(* IEC 61131-3 sources: intralogisticsai/plc_programs, 4 files *)

(* ---- roots_warehouse_simulation.st ---- *)
PROGRAM RootsWarehouseSimulation
  VAR
    (* Physical I/O *)
    emergency_stop AT %IX0.0 : BOOL;
    manual_reset AT %IX0.1 : BOOL;

    (* Process Control Signals - MODBUS 1000-1008 *)
    plc_cycle_stopped AT %QX125.0 : BOOL;
    plc_cycle_running AT %QX125.1 : BOOL;
    pick_error AT %QX125.2 : BOOL;
    pick_to_assembly_in_process AT %QX125.3 : BOOL;
    pick_to_assembly_complete AT %QX125.4 : BOOL;
    pick_to_receiving_in_process AT %QX125.5 : BOOL;
    pick_to_receiving_complete AT %QX125.6 : BOOL;
    pick_to_warehouse_in_process AT %QX125.7 : BOOL;
    pick_to_warehouse_complete AT %QX126.0 : BOOL;

    (* Pick Bin Controls - MODBUS 2000-2011 - ERP Controlled Coils *)
    pick_bin_01 AT %QX250.0 : BOOL;
    pick_bin_02 AT %QX250.1 : BOOL;
    pick_bin_03 AT %QX250.2 : BOOL;
    pick_bin_04 AT %QX250.3 : BOOL;
    pick_bin_05 AT %QX250.4 : BOOL;
    pick_bin_06 AT %QX250.5 : BOOL;
    pick_bin_07 AT %QX250.6 : BOOL;
    pick_bin_08 AT %QX250.7 : BOOL;
    pick_bin_09 AT %QX251.0 : BOOL;
    pick_bin_10 AT %QX251.1 : BOOL;
    pick_bin_11 AT %QX251.2 : BOOL;
    pick_bin_12 AT %QX251.3 : BOOL;

    (* Station Status Controls - MODBUS 2020-2023 - ERP Controlled Coils *)
    to_receiving_sta_1 AT %QX252.4 : BOOL;
    from_receiving_sta_1 AT %QX252.5 : BOOL;
    to_assembly_sta_2 AT %QX252.6 : BOOL;
    from_assembly_sta_2 AT %QX252.7 : BOOL;

    (* Statistics and Monitoring - MODBUS 100-106 *)
    cycle_counter AT %MW100 : INT;
    pick_operations_total AT %MW101 : INT;
    assembly_picks AT %MW102 : INT;
    receiving_picks AT %MW103 : INT;
    warehouse_picks AT %MW104 : INT;
    error_count AT %MW105 : INT;
    uptime_seconds AT %MW106 : INT;
END_VAR

VAR
    (* Internal Variables - No direct addressing *)
    assembly_timer : INT;
    receiving_timer : INT;
    warehouse_timer : INT;
    assembly_complete_timer : INT;
    receiving_complete_timer : INT;
    warehouse_complete_timer : INT;
    any_bin_selected : BOOL;
    assembly_requested : BOOL;
    receiving_requested : BOOL;
    warehouse_requested : BOOL;
    assembly_in_progress : BOOL;
    receiving_in_progress : BOOL;
    warehouse_in_progress : BOOL;
    uptime_timer : INT;
END_VAR

(* Perfect world system - always running, never errors *)
  plc_cycle_running := TRUE;
  plc_cycle_stopped := FALSE;
  pick_error := FALSE;

  (* Increment counters *)
  cycle_counter := cycle_counter + 1;

  (* Uptime calculation - increment every 10 cycles (approximately 1 second at 100ms) *)
  uptime_timer := uptime_timer + 1;
  IF uptime_timer >= 10 THEN
    uptime_timer := 0;
    uptime_seconds := uptime_seconds + 1;
  END_IF;

  (* ERP Command Detection *)
  any_bin_selected := pick_bin_01 OR pick_bin_02 OR pick_bin_03 OR pick_bin_04 OR pick_bin_05 OR pick_bin_06 OR pick_bin_07 OR pick_bin_08 OR pick_bin_09 OR pick_bin_10 OR pick_bin_11 OR pick_bin_12;

  assembly_requested := any_bin_selected AND to_assembly_sta_2;
  receiving_requested := any_bin_selected AND to_receiving_sta_1;
  warehouse_requested := any_bin_selected AND (NOT to_assembly_sta_2) AND (NOT to_receiving_sta_1);

  (* Assembly Operation - 20 Second Robot Simulation *)
  IF assembly_requested AND NOT assembly_in_progress THEN
    (* Start assembly operation *)
    assembly_in_progress := TRUE;
    pick_to_assembly_in_process := TRUE;
    assembly_timer := 0;
  END_IF;

  IF assembly_in_progress THEN
    assembly_timer := assembly_timer + 1;
    IF assembly_timer >= 200 THEN (* 20.0 seconds at 100ms cycles *)
      (* Complete assembly operation *)
      pick_to_assembly_complete := TRUE;
      pick_to_assembly_in_process := FALSE;
      assembly_in_progress := FALSE;
      assembly_timer := 0;
      assembly_picks := assembly_picks + 1;
      pick_operations_total := pick_operations_total + 1;
    END_IF;
  END_IF;

  (* Receiving Operation - 20 Second Robot Simulation *)
  IF receiving_requested AND NOT receiving_in_progress THEN
    (* Start receiving operation *)
    receiving_in_progress := TRUE;
    pick_to_receiving_in_process := TRUE;
    receiving_timer := 0;
  END_IF;

  IF receiving_in_progress THEN
    receiving_timer := receiving_timer + 1;
    IF receiving_timer >= 200 THEN (* 20.0 seconds at 100ms cycles *)
      (* Complete receiving operation *)
      pick_to_receiving_complete := TRUE;
      pick_to_receiving_in_process := FALSE;
      receiving_in_progress := FALSE;
      receiving_timer := 0;
      receiving_picks := receiving_picks + 1;
      pick_operations_total := pick_operations_total + 1;
    END_IF;
  END_IF;

  (* Warehouse Operation - 20 Second Robot Simulation *)
  IF warehouse_requested AND NOT warehouse_in_progress THEN
    (* Start warehouse operation *)
    warehouse_in_progress := TRUE;
    pick_to_warehouse_in_process := TRUE;
    warehouse_timer := 0;
  END_IF;

  IF warehouse_in_progress THEN
    warehouse_timer := warehouse_timer + 1;
    IF warehouse_timer >= 200 THEN (* 20.0 seconds at 100ms cycles *)
      (* Complete warehouse operation *)
      pick_to_warehouse_complete := TRUE;
      pick_to_warehouse_in_process := FALSE;
      warehouse_in_progress := FALSE;
      warehouse_timer := 0;
      warehouse_picks := warehouse_picks + 1;
      pick_operations_total := pick_operations_total + 1;
    END_IF;
  END_IF;

  (* Auto-reset COMPLETE signals after 10 seconds to allow ERP processing time *)
  IF pick_to_assembly_complete THEN
    assembly_complete_timer := assembly_complete_timer + 1;
    IF assembly_complete_timer >= 100 THEN (* 10 seconds *)
      pick_to_assembly_complete := FALSE;
      assembly_complete_timer := 0;
    END_IF;
  ELSE
    assembly_complete_timer := 0;
  END_IF;

  IF pick_to_receiving_complete THEN
    receiving_complete_timer := receiving_complete_timer + 1;
    IF receiving_complete_timer >= 100 THEN (* 10 seconds *)
      pick_to_receiving_complete := FALSE;
      receiving_complete_timer := 0;
    END_IF;
  ELSE
    receiving_complete_timer := 0;
  END_IF;

  IF pick_to_warehouse_complete THEN
    warehouse_complete_timer := warehouse_complete_timer + 1;
    IF warehouse_complete_timer >= 100 THEN (* 10 seconds *)
      pick_to_warehouse_complete := FALSE;
      warehouse_complete_timer := 0;
    END_IF;
  ELSE
    warehouse_complete_timer := 0;
  END_IF;

END_PROGRAM

CONFIGURATION Config0
  RESOURCE Res0 ON PLC
    TASK Main(INTERVAL := T#100ms,PRIORITY := 0);
    PROGRAM Inst0 WITH Main : RootsWarehouseSimulation;
  END_RESOURCE
END_CONFIGURATION

(* ---- simple_modbus_server.st ---- *)
(*
Simple CODESYS Structured Text Program
Intralogistics Learning Lab - Basic MODBUS TCP Server
Provides basic I/O simulation compatible with ERP integration
*)

PROGRAM PLC_PRG
VAR
    (* Conveyor System Variables *)
    Conveyor1_Run: BOOL := FALSE;           (* Address 40001 *)
    Conveyor1_Speed: INT := 0;              (* Address 40002 *)
    Conveyor1_Status: BOOL := FALSE;        (* Address 40003 *)

    Conveyor2_Run: BOOL := FALSE;           (* Address 40004 *)
    Conveyor2_Speed: INT := 0;              (* Address 40005 *)
    Conveyor2_Status: BOOL := FALSE;        (* Address 40006 *)

    (* Storage Robot Variables *)
    Robot_Position_X: INT := 0;             (* Address 40007 *)
    Robot_Position_Y: INT := 0;             (* Address 40008 *)
    Robot_Position_Z: INT := 0;             (* Address 40009 *)
    Robot_Gripper_Open: BOOL := FALSE;      (* Address 40010 *)
    Robot_Busy: BOOL := FALSE;              (* Address 40011 *)

    (* RFID System Variables *)
    RFID_Station1_Active: BOOL := FALSE;    (* Address 40012 *)
    RFID_Station1_TagID: DWORD := 0;        (* Address 40013-40014 *)
    RFID_Station2_Active: BOOL := FALSE;    (* Address 40015 *)
    RFID_Station2_TagID: DWORD := 0;        (* Address 40016-40017 *)

    (* Safety System *)
    Emergency_Stop: BOOL := FALSE;          (* Address 40018 *)
    Safety_OK: BOOL := TRUE;                (* Address 40019 *)
    System_Ready: BOOL := FALSE;            (* Address 40020 *)

    (* Simulation Timers *)
    Cycle_Timer: TIME;
    Robot_Move_Timer: TIME;

    (* Internal simulation variables *)
    Simulation_Active: BOOL := TRUE;
    Cycle_Count: INT := 0;
END_VAR

(* Main Program Logic *)

(* System Ready Logic *)
System_Ready := Safety_OK AND NOT Emergency_Stop;

(* Conveyor Control Logic *)
IF System_Ready THEN
    IF Conveyor1_Run THEN
        Conveyor1_Status := TRUE;
        IF Conveyor1_Speed = 0 THEN
            Conveyor1_Speed := 50;  (* Default speed *)
        END_IF
    ELSE
        Conveyor1_Status := FALSE;
        Conveyor1_Speed := 0;
    END_IF

    IF Conveyor2_Run THEN
        Conveyor2_Status := TRUE;
        IF Conveyor2_Speed = 0 THEN
            Conveyor2_Speed := 50;  (* Default speed *)
        END_IF
    ELSE
        Conveyor2_Status := FALSE;
        Conveyor2_Speed := 0;
    END_IF
ELSE
    (* Emergency stop - halt all conveyors *)
    Conveyor1_Status := FALSE;
    Conveyor1_Speed := 0;
    Conveyor2_Status := FALSE;
    Conveyor2_Speed := 0;
END_IF

(* Robot Simulation Logic *)
IF System_Ready AND NOT Robot_Busy THEN
    (* Simple position simulation *)
    IF Cycle_Count MOD 100 = 0 THEN
        Robot_Position_X := Robot_Position_X + 10;
        IF Robot_Position_X > 1000 THEN
            Robot_Position_X := 0;
        END_IF
    END_IF

    IF Cycle_Count MOD 150 = 0 THEN
        Robot_Position_Y := Robot_Position_Y + 5;
        IF Robot_Position_Y > 500 THEN
            Robot_Position_Y := 0;
        END_IF
    END_IF

    (* Gripper simulation *)
    IF Cycle_Count MOD 200 = 0 THEN
        Robot_Gripper_Open := NOT Robot_Gripper_Open;
    END_IF
END_IF

(* RFID Simulation Logic *)
IF System_Ready THEN
    IF Cycle_Count MOD 300 = 0 THEN
        RFID_Station1_Active := NOT RFID_Station1_Active;
        IF RFID_Station1_Active THEN
            RFID_Station1_TagID := RFID_Station1_TagID + 1;
            IF RFID_Station1_TagID = 0 THEN
                RFID_Station1_TagID := 1000;  (* Start from 1000 *)
            END_IF
        END_IF
    END_IF

    IF Cycle_Count MOD 350 = 0 THEN
        RFID_Station2_Active := NOT RFID_Station2_Active;
        IF RFID_Station2_Active THEN
            RFID_Station2_TagID := RFID_Station2_TagID + 1;
            IF RFID_Station2_TagID = 0 THEN
                RFID_Station2_TagID := 2000;  (* Start from 2000 *)
            END_IF
        END_IF
    END_IF
END_IF

(* Cycle counter for simulation timing *)
Cycle_Count := Cycle_Count + 1;
IF Cycle_Count > 32000 THEN
    Cycle_Count := 0;
END_IF

END_PROGRAM

(*
MODBUS TCP Server Configuration:
- Port: 502
- Unit ID: 1
- Function Codes: 3 (Read Holding Registers), 6 (Write Single Register), 16 (Write Multiple Registers)

Register Map:
40001: Conveyor1_Run (BOOL)
40002: Conveyor1_Speed (INT)
40003: Conveyor1_Status (BOOL)
40004: Conveyor2_Run (BOOL)
40005: Conveyor2_Speed (INT)
40006: Conveyor2_Status (BOOL)
40007: Robot_Position_X (INT)
40008: Robot_Position_Y (INT)
40009: Robot_Position_Z (INT)
40010: Robot_Gripper_Open (BOOL)
40011: Robot_Busy (BOOL)
40012: RFID_Station1_Active (BOOL)
40013-40014: RFID_Station1_TagID (DWORD)
40015: RFID_Station2_Active (BOOL)
40016-40017: RFID_Station2_TagID (DWORD)
40018: Emergency_Stop (BOOL)
40019: Safety_OK (BOOL)
40020: System_Ready (BOOL)
*)

(* ---- simple_modbus_test.st ---- *)
PROGRAM PLC_PRG
VAR
    ModbusSlaveRequestHandler_TCP: ModbusSlaveRequestHandler_TCP;
    ServerStatus: BOOL := FALSE;
    TestCounter: UINT := 0;

    (* Test coils for bin selection *)
    Bin01_Selected AT %QX100.0: BOOL;
    Bin02_Selected AT %QX100.1: BOOL;
    Bin03_Selected AT %QX100.2: BOOL;
    Bin04_Selected AT %QX100.3: BOOL;

    (* Test registers *)
    SystemStatus AT %QW200: UINT;
    RobotPosition AT %QW201: UINT;
END_VAR

(* Main program loop *)
TestCounter := TestCounter + 1;
IF TestCounter > 1000 THEN
    TestCounter := 0;
END_IF

(* Update test registers *)
SystemStatus := 1; (* System running *)
RobotPosition := TestCounter;

(* Simple MODBUS TCP server *)
ModbusSlaveRequestHandler_TCP(
    Enable := TRUE,
    Address := '0.0.0.0',
    Port := 502,
    pMemoryArea := ADR(%MB0),
    uiMemoryAreaSize := 1000
);

ServerStatus := ModbusSlaveRequestHandler_TCP.xReady;

(* ---- traffic_light_controller.st ---- *)
PROGRAM traffic_light_controller
VAR
    pedestrian_ns_button AT %IX0.0 : BOOL;
    pedestrian_ew_button AT %IX0.1 : BOOL;
    emergency_override AT %IX0.2 : BOOL;
    system_enable AT %IX0.3 : BOOL;
    manual_reset AT %IX0.4 : BOOL;

    ns_red_light AT %QX0.0 : BOOL;
    ns_yellow_light AT %QX0.1 : BOOL;
    ns_green_light AT %QX0.2 : BOOL;
    ew_red_light AT %QX0.3 : BOOL;
    ew_yellow_light AT %QX0.4 : BOOL;
    ew_green_light AT %QX0.5 : BOOL;
    ped_ns_walk AT %QX0.6 : BOOL;
    ped_ns_dont_walk AT %QX0.7 : BOOL;
    ped_ew_walk AT %QX1.0 : BOOL;
    ped_ew_dont_walk AT %QX1.1 : BOOL;

    system_state AT %MW0 : INT;
    ns_green_cycles AT %MW1 : INT;
    ew_green_cycles AT %MW2 : INT;
    ped_ns_cycles AT %MW3 : INT;
    ped_ew_cycles AT %MW4 : INT;
    emergency_activations AT %MW5 : INT;
    total_runtime_seconds AT %MW6 : INT;

    timer_main : TON;
    timer_yellow : TON;
    timer_ped : TON;
    timer_emergency : TON;
    runtime_timer : TON;

    green_time_ns : TIME := T#30000MS;
    green_time_ew : TIME := T#25000MS;
    yellow_time : TIME := T#5000MS;
    ped_walk_time : TIME := T#15000MS;
    ped_clear_time : TIME := T#10000MS;
    emergency_flash_time : TIME := T#500MS;

    STATE_NS_GREEN : INT := 1;
    STATE_NS_YELLOW : INT := 2;
    STATE_EW_GREEN : INT := 3;
    STATE_EW_YELLOW : INT := 4;
    STATE_PED_NS_WALK : INT := 5;
    STATE_PED_NS_CLEAR : INT := 6;
    STATE_PED_EW_WALK : INT := 7;
    STATE_PED_EW_CLEAR : INT := 8;
    STATE_EMERGENCY : INT := 9;

    ped_ns_request : BOOL := FALSE;
    ped_ew_request : BOOL := FALSE;
    emergency_active : BOOL := FALSE;
    emergency_flash_state : BOOL := FALSE;

    ped_ns_btn_prev : BOOL := FALSE;
    ped_ew_btn_prev : BOOL := FALSE;
    emergency_btn_prev : BOOL := FALSE;

    system_running : BOOL;
    emergency_mode : BOOL;
    fault_status : BOOL;

    cycle_count_total : INT;
    avg_cycle_time : INT;
    last_emergency_time : TIME;
END_VAR

(* Main Program Logic *)

(* Initialize system on first run *)
IF system_state = 0 AND system_enable THEN
    system_state := STATE_NS_GREEN;
    ns_green_cycles := 0;
    ew_green_cycles := 0;
    ped_ns_cycles := 0;
    ped_ew_cycles := 0;
    emergency_activations := 0;
    total_runtime_seconds := 0;
END_IF;

(* Runtime Counter - Increment every second *)
runtime_timer(IN:=system_enable, PT:=T#1000MS);
IF runtime_timer.Q THEN
    runtime_timer(IN:=FALSE);
    runtime_timer(IN:=TRUE);
    total_runtime_seconds := total_runtime_seconds + 1;
END_IF;

(* Edge Detection for Pedestrian Buttons *)
IF pedestrian_ns_button AND NOT ped_ns_btn_prev THEN
    ped_ns_request := TRUE;
END_IF;
ped_ns_btn_prev := pedestrian_ns_button;

IF pedestrian_ew_button AND NOT ped_ew_btn_prev THEN
    ped_ew_request := TRUE;
END_IF;
ped_ew_btn_prev := pedestrian_ew_button;

(* Edge Detection for Emergency Override *)
IF emergency_override AND NOT emergency_btn_prev THEN
    emergency_active := TRUE;
    emergency_activations := emergency_activations + 1;
    (* last_emergency_time := current_time; *)
END_IF;
emergency_btn_prev := emergency_override;

(* Emergency Override Logic *)
IF emergency_active AND emergency_override THEN
    system_state := STATE_EMERGENCY;
    emergency_mode := TRUE;
ELSIF emergency_active AND NOT emergency_override THEN
    emergency_active := FALSE;
    emergency_mode := FALSE;
    system_state := STATE_NS_GREEN;
    timer_main(IN:=FALSE);
END_IF;

(* Manual Reset *)
IF manual_reset THEN
    system_state := STATE_NS_GREEN;
    ped_ns_request := FALSE;
    ped_ew_request := FALSE;
    emergency_active := FALSE;
    emergency_mode := FALSE;
    timer_main(IN:=FALSE);
    timer_yellow(IN:=FALSE);
    timer_ped(IN:=FALSE);
    timer_emergency(IN:=FALSE);
END_IF;

(* Main State Machine *)
CASE system_state OF

    STATE_NS_GREEN:
        (* North-South Green Light *)
        ns_red_light := FALSE;
        ns_yellow_light := FALSE;
        ns_green_light := TRUE;
        ew_red_light := TRUE;
        ew_yellow_light := FALSE;
        ew_green_light := FALSE;

        (* Pedestrian Signals *)
        ped_ns_walk := FALSE;
        ped_ns_dont_walk := TRUE;
        ped_ew_walk := FALSE;
        ped_ew_dont_walk := TRUE;

        (* Timer for green phase *)
        timer_main(IN:=TRUE, PT:=green_time_ns);

        IF timer_main.Q THEN
            timer_main(IN:=FALSE);
            ns_green_cycles := ns_green_cycles + 1;
            cycle_count_total := cycle_count_total + 1;

            (* Check for pedestrian request *)
            IF ped_ew_request THEN
                system_state := STATE_PED_EW_WALK;
                ped_ew_request := FALSE;
            ELSE
                system_state := STATE_NS_YELLOW;
            END_IF;
        END_IF;

    STATE_NS_YELLOW:
        (* North-South Yellow Light *)
        ns_red_light := FALSE;
        ns_yellow_light := TRUE;
        ns_green_light := FALSE;
        ew_red_light := TRUE;
        ew_yellow_light := FALSE;
        ew_green_light := FALSE;

        timer_yellow(IN:=TRUE, PT:=yellow_time);

        IF timer_yellow.Q THEN
            timer_yellow(IN:=FALSE);
            system_state := STATE_EW_GREEN;
        END_IF;

    STATE_EW_GREEN:
        (* East-West Green Light *)
        ns_red_light := TRUE;
        ns_yellow_light := FALSE;
        ns_green_light := FALSE;
        ew_red_light := FALSE;
        ew_yellow_light := FALSE;
        ew_green_light := TRUE;

        (* Pedestrian Signals *)
        ped_ns_walk := FALSE;
        ped_ns_dont_walk := TRUE;
        ped_ew_walk := FALSE;
        ped_ew_dont_walk := TRUE;

        timer_main(IN:=TRUE, PT:=green_time_ew);

        IF timer_main.Q THEN
            timer_main(IN:=FALSE);
            ew_green_cycles := ew_green_cycles + 1;
            cycle_count_total := cycle_count_total + 1;

            (* Check for pedestrian request *)
            IF ped_ns_request THEN
                system_state := STATE_PED_NS_WALK;
                ped_ns_request := FALSE;
            ELSE
                system_state := STATE_EW_YELLOW;
            END_IF;
        END_IF;

    STATE_EW_YELLOW:
        (* East-West Yellow Light *)
        ns_red_light := TRUE;
        ns_yellow_light := FALSE;
        ns_green_light := FALSE;
        ew_red_light := FALSE;
        ew_yellow_light := TRUE;
        ew_green_light := FALSE;

        timer_yellow(IN:=TRUE, PT:=yellow_time);

        IF timer_yellow.Q THEN
            timer_yellow(IN:=FALSE);
            system_state := STATE_NS_GREEN;
        END_IF;

    STATE_PED_NS_WALK:
        (* Pedestrian North-South Walk Phase *)
        ns_red_light := TRUE;
        ns_yellow_light := FALSE;
        ns_green_light := FALSE;
        ew_red_light := TRUE;
        ew_yellow_light := FALSE;
        ew_green_light := FALSE;

        ped_ns_walk := TRUE;
        ped_ns_dont_walk := FALSE;
        ped_ew_walk := FALSE;
        ped_ew_dont_walk := TRUE;

        timer_ped(IN:=TRUE, PT:=ped_walk_time);

        IF timer_ped.Q THEN
            timer_ped(IN:=FALSE);
            ped_ns_cycles := ped_ns_cycles + 1;
            system_state := STATE_PED_NS_CLEAR;
        END_IF;

    STATE_PED_NS_CLEAR:
        (* Pedestrian North-South Clearance Phase *)
        ns_red_light := TRUE;
        ns_yellow_light := FALSE;
        ns_green_light := FALSE;
        ew_red_light := TRUE;
        ew_yellow_light := FALSE;
        ew_green_light := FALSE;

        ped_ns_walk := FALSE;
        ped_ns_dont_walk := TRUE;
        ped_ew_walk := FALSE;
        ped_ew_dont_walk := TRUE;

        timer_ped(IN:=TRUE, PT:=ped_clear_time);

        IF timer_ped.Q THEN
            timer_ped(IN:=FALSE);
            system_state := STATE_EW_GREEN;
        END_IF;

    STATE_PED_EW_WALK:
        (* Pedestrian East-West Walk Phase *)
        ns_red_light := TRUE;
        ns_yellow_light := FALSE;
        ns_green_light := FALSE;
        ew_red_light := TRUE;
        ew_yellow_light := FALSE;
        ew_green_light := FALSE;

        ped_ns_walk := FALSE;
        ped_ns_dont_walk := TRUE;
        ped_ew_walk := TRUE;
        ped_ew_dont_walk := FALSE;

        timer_ped(IN:=TRUE, PT:=ped_walk_time);

        IF timer_ped.Q THEN
            timer_ped(IN:=FALSE);
            ped_ew_cycles := ped_ew_cycles + 1;
            system_state := STATE_PED_EW_CLEAR;
        END_IF;

    STATE_PED_EW_CLEAR:
        (* Pedestrian East-West Clearance Phase *)
        ns_red_light := TRUE;
        ns_yellow_light := FALSE;
        ns_green_light := FALSE;
        ew_red_light := TRUE;
        ew_yellow_light := FALSE;
        ew_green_light := FALSE;

        ped_ns_walk := FALSE;
        ped_ns_dont_walk := TRUE;
        ped_ew_walk := FALSE;
        ped_ew_dont_walk := TRUE;

        timer_ped(IN:=TRUE, PT:=ped_clear_time);

        IF timer_ped.Q THEN
            timer_ped(IN:=FALSE);
            system_state := STATE_NS_GREEN;
        END_IF;

    STATE_EMERGENCY:
        (* Emergency Mode - Flash All Red *)
        timer_emergency(IN:=TRUE, PT:=emergency_flash_time);

        IF timer_emergency.Q THEN
            timer_emergency(IN:=FALSE);
            emergency_flash_state := NOT emergency_flash_state;
        END_IF;

        IF emergency_flash_state THEN
            ns_red_light := TRUE;
            ns_yellow_light := FALSE;
            ns_green_light := FALSE;
            ew_red_light := TRUE;
            ew_yellow_light := FALSE;
            ew_green_light := FALSE;
        ELSE
            ns_red_light := FALSE;
            ns_yellow_light := FALSE;
            ns_green_light := FALSE;
            ew_red_light := FALSE;
            ew_yellow_light := FALSE;
            ew_green_light := FALSE;
        END_IF;

        (* Pedestrian signals off during emergency *)
        ped_ns_walk := FALSE;
        ped_ns_dont_walk := emergency_flash_state;
        ped_ew_walk := FALSE;
        ped_ew_dont_walk := emergency_flash_state;

END_CASE;

(* System Status *)
system_running := system_enable AND (system_state > 0);
fault_status := NOT system_enable OR (system_state = 0);

(* Calculate Average Cycle Time *)
IF cycle_count_total > 0 THEN
    avg_cycle_time := total_runtime_seconds / cycle_count_total;
ELSE
    avg_cycle_time := 0;
END_IF;

END_PROGRAM
